{attribute 'qualified_only'}
{attribute 'strict'}
TYPE E_LogLevel :
(
	eTrace 	:= 0,
	eDebug 	:= 1,
	eInfo	:= 2,
	eWarn	:= 3,
	eError	:= 4,
	eFatal	:= 5
) UINT;
END_TYPE

(* stored: Version 1.1.0.1, ProductVersion 3.1.4024.0
   DUT E_LogLevel: Id {322cf33f-cf60-45fe-86fc-20e9e85b0465} *)
